Fanuc KAREL source: ko00142.KL

-- PROVISIONAL review KL for V770-1; original PC SHA256 77f14453779af369698930cf167ec7aec691451a78a9f8b93d75d448b9872d74
-- Incomplete behavior may be omitted. Consult companion uncertainty JSON. Do not deploy.
PROGRAM KO00142
%NOLOCKGROUP
VAR
  R : REAL
  N : REAL
-- UNRESOLVED_DECL CFG type=00001c
-- UNRESOLVED_DECL OUT type=000102
BEGIN
  -- UNRESOLVED_PC offsets 5-13; opcodes 9D,64,23
  -- UNRESOLVED_PC offsets 18-29; opcodes 2E,23
  -- UNRESOLVED_PC offsets 34-44; opcodes 9D,22,A5
  -- UNRESOLVED_PC offsets 49-106; opcodes 27,22,22,22,22,22,22,22,76,7E,4A
  -- UNRESOLVED_PC offsets 111-115; opcodes 7F
END KO00142
